TYPE EL6002_Control :
STRUCT
	{attribute addProperty Name "Transmit request"}
	TransmitRequest : BIT;
	{attribute addProperty Name "Receive accepted"}
	ReceiveAccepted : BIT;
	{attribute addProperty Name "Init request"}
	InitRequest : BIT;
	{attribute addProperty Name "Send continues"}
	SendContinues : BIT;
	{attribute 'hide'}
	{attribute addProperty Name "Bit 5(address x.4)"}
	Bit_5 : BIT;
	{attribute 'hide'}
	{attribute addProperty Name "Bit 6(address x.5)"}
	Bit_6 : BIT;
	{attribute 'hide'}
	{attribute addProperty Name "Bit 7(address x.6)"}
	Bit_7 : BIT;
	{attribute 'hide'}
	{attribute addProperty Name "Bit 8(address x.7)"}
	Bit_8 : BIT;
	{attribute addProperty Name "Output length"}
	OutputLength : USINT;
END_STRUCT
END_TYPE

(* stored: Version 1.1.0.1, ProductVersion 3.1.4024.9
   DUT EL6002_Control: Id {f13b5f51-2661-0b9e-1dd3-dd6d48761ebe} *)
